/// Abstract base FB for components
{attribute 'reflection' := ''}
FUNCTION_BLOCK ABSTRACT FB_Component IMPLEMENTS ITF_Component

VAR
	/// path of this FB
	{attribute 'no_init' := ''}
	{attribute 'instance-path' := ''}
	sPath						: STRING;	
	/// Unique ID
	nId							: INT;		
	/// component type
	eTyp						: E_ComponentType;
	/// component name
	sName						: STRING;
	/// BMK name
	sBMK						: STRING;
	/// Area
	eMachineArea				: E_MachineArea;			
	
	/// component enable flag
	bEnable						: BOOL := FALSE;
	/// component state
	eState						: E_ComponentState;	
	
	/// Safety
	refEStop					: REFERENCE TO FB_EmergencyStop;
	aitfSafetyComp				: ARRAY[0..COMP.nMaxComponents] OF ITF_SafetyComp;
	bAccessPermit				: BOOL;


	/// Others
	itfEventLog					: ITF_EventLog;
	refSetting					: REFERENCE TO ST_MachineSetting;

	nChangeToggle				: INT;
END_VAR

///
/// 
/// HF/www.asma.at/02.2022
///

PROPERTY AccessPermit : BOOL
GET
AccessPermit := bAccessPermit;
END_GET
END_PROPERTY

/// RunSuper component logic
{attribute 'object_name' := 'Base'}
METHOD Base

VAR
	ni			: INT;
END_VAR
// DEFAULT STATE: set state to running
IF eState = E_ComponentState.ready THEN
	eState := E_ComponentState.running;
END_IF

//Eventlog
IF itfEventLog = 0 THEN
	WriteError(E_Event.eEvent_none, 'HMI Referenz nicht gesetzt!');
	eState := E_ComponentState.error;
	RETURN;
END_IF


Visu();

IF NOT Enable THEN
	RETURN;
END_IF

Run();
END_METHOD

PROPERTY BMK : STRING
GET
BMK := sBMK;
END_GET
SET
sBMK := BMK;
END_SET
END_PROPERTY

METHOD ChangeToggle : BOOL
VAR_INPUT
END_VAR
nChangeToggle := nChangeToggle + 1;
END_METHOD

PROPERTY EmergencyStop : REFERENCE TO FB_EmergencyStop
GET
IF __ISVALIDREF(refEStop) THEN
	EmergencyStop REF= refEStop;
END_IF
END_GET
SET
refEStop REF= EmergencyStop;
END_SET
END_PROPERTY

/// Get's or set's a value indicating whether this component is active or not.
PROPERTY Enable : BOOL
GET
Enable := bEnable;
END_GET
SET
bEnable := Enable;
END_SET
END_PROPERTY

METHOD FB_init : BOOL
VAR_INPUT
	bInitRetains : BOOL := TRUE; // if TRUE, the retain variables are initialized (warm start / cold start)
	bInCopyCode : BOOL := TRUE;  // if TRUE, the instance afterwards gets moved into the copy code (online change)
END_VAR
nId := nId + 1;
itfEventLog := GVL.fbEventLog;
refSetting REF= GVL.stSetting;
refEStop REF= GVL.fbEStop;
Init();
END_METHOD

/// Halt component logic
{attribute 'object_name' := 'Halt'}
METHOD Halt : E_OperationResult

VAR_INPUT
	StoppCategory					: INT;			// 0...ungesteuertes Stillsetzen     1...gesteuertes Stillsetzen     2...gesteuertes Stillsetzen ohne Trennung der Energiezufuhr							
END_VAR
bAccessPermit := TRUE;
END_METHOD

/// Unique component ID (cam be used as index: P_ComponentPool.aComponents[eID]...)
PROPERTY ID : INT
GET
ID := nId;
END_GET
SET
nId := Id;
END_SET
END_PROPERTY

/// Init component logic
{attribute 'object_name' := 'Init'}
METHOD Init : E_OperationResult
END_METHOD

PROPERTY MachineArea : E_MachineArea
GET
MachineArea := eMachineArea;
END_GET
SET
eMachineArea := MachineArea;
END_SET
END_PROPERTY

PROPERTY Name : STRING
GET
Name := sName;
END_GET
SET
sName := Name;
END_SET
END_PROPERTY

PROPERTY Path : String
GET
Path := sPath;
END_GET
END_PROPERTY

METHOD RegisterSafetyComp : BOOL
VAR_INPUT
	SafetyComp				: ITF_SafetyComp;
END_VAR
VAR
	ni						: INT;
END_VAR
FOR ni:= 0 TO COMP.nMaxComponents DO

	IF aitfSafetyComp[ni] = SafetyComp THEN
		RETURN;
	END_IF
	
	IF aitfSafetyComp[ni] <> 0 THEN
		CONTINUE;
	END_IF
	
	aitfSafetyComp[ni] := SafetyComp;
	aitfSafetyComp[ni].RegisterComponent(THIS^);
	RETURN;
	
END_FOR
END_METHOD

/// ResetSuper component logic
{attribute 'object_name' := 'Reset'}
METHOD Reset : E_OperationResult
// DEFAULT STATE: set state to ready
eState := E_ComponentState.ready;
END_METHOD

/// RestartSuper component logic
{attribute 'object_name' := 'Restart'}
METHOD Restart : E_OperationResult
VAR_INPUT
END_VAR
bAccessPermit := FALSE;
END_METHOD

/// RunSuper component logic
{attribute 'object_name' := 'Run'}
METHOD Abstract Run
END_METHOD

PROPERTY SafeEnvironment : BOOL
GET
VAR
	ni				: INT;
END_VAR
SafeEnvironment := TRUE;

FOR ni:= 0 TO COMP.nMaxComponents DO
	
	IF aitfSafetyComp[ni] <> 0 AND_THEN NOT aitfSafetyComp[ni].Safe THEN
		SafeEnvironment := FALSE;
	END_IF

END_FOR
END_GET
END_PROPERTY

/// Get's value representing the component state.
PROPERTY State : E_ComponentState
GET
State := eState;
END_GET
END_PROPERTY

/// Get's value representing the component state.
PROPERTY StateAsString : STRING
GET
CASE eState OF

	E_ComponentState.none :
		StateAsString := 'undefiniert';
	/// Component is resetting
	E_ComponentState.resetting:
		StateAsString := 'wird zurückgesetzt';
	/// Component is ready
	E_ComponentState.ready:
		StateAsString := 'ist bereit';
	/// Component is running
	E_ComponentState.running:
		StateAsString := 'wird ausgeführt';
	/// Component has error
	E_ComponentState.error:
		StateAsString := 'ist fehlerhaft';

END_CASE
END_GET
END_PROPERTY

PROPERTY Typ : E_ComponentType
GET
Typ := eTyp;
END_GET
END_PROPERTY

/// Visu component logic
{attribute 'object_name' := 'Visu'}
METHOD Abstract Visu
END_METHOD

METHOD VisuBase
VAR_IN_OUT
	stCompVisu					: ST_ComponentVisu;
END_VAR
// Visu
stCompVisu.bEnable := bEnable;
stCompVisu.bAccessPermit := AccessPermit;
stCompVisu.bError := eState = E_Componentstate.error;
stCompVisu.bRunning := eState = E_Componentstate.running;
stCompVisu.eState := eState;
stCompVisu.sName := sName;

IF stCompVisu.bReset THEN
	stCompVisu.bReset := FALSE;	
	Reset();
END_IF
END_METHOD

METHOD WriteError
VAR_INPUT
	Event			: E_Event;
	Description 	: T_MaxString;
END_VAR
WriteEvent(ePriority_fault, Event, Description, TRUE);
END_METHOD

METHOD WriteEvent
VAR_INPUT
	Priority		: E_Priority;
	Event			: E_Event;
	Description 	: T_MaxString;
	Signalize		: BOOL;
END_VAR
VAR
	tmpItem: ST_Event;
END_VAR
// chk
IF itfEventLog = 0 THEN
	RETURN;
END_IF

tmpItem.eComponent := eTyp;
tmpItem.eEventID := Event;
tmpItem.eMachineArea := eMachineArea;
tmpItem.sPosition := sBMK;
tmpItem.ePriority := Priority;
tmpItem.nComponentID := nId;
tmpItem.sDescription := Description;
tmpItem.bSignalize := Signalize;
tmpItem.refComponent REF= THIS^;

itfEventLog.SetEvent(tmpItem);
END_METHOD

METHOD WriteInfo
VAR_INPUT
	Event			: E_Event;
	Description 	: T_MaxString;
END_VAR
WriteEvent(ePriority_info, Event, Description, FALSE);
END_METHOD

METHOD WriteWarning
VAR_INPUT
	Event			: E_Event;
	Description 	: T_MaxString;
	Signal			: BOOL;
END_VAR
VAR
	tmpItem			: ST_Event;
END_VAR
WriteEvent(ePriority_warning, Event, Description, Signal);
END_METHOD

END_FUNCTION_BLOCK

(* stored: Version 1.1.0.1
   POU FB_Component: Id {c18f24bd-a664-4b00-87c6-35388a9e2c13}, SpecialFunc None
   Folder Abstract: Id {74ace20b-84be-4a97-82c0-d348ab638f2b}
   Folder Properties: Id {2d8306c8-917b-4b20-9aa7-5415be6cad83}
   Folder Utilities: Id {18cd2ad0-5a5a-4e5f-92e4-b0238b542ab5}
   Property AccessPermit: Id {01de2613-1fdc-4238-9d0f-b61744631c69}
   Get Get: Id {d0f0ca6c-2e80-4b7b-abfc-89db46355afd}
   Method Base: Id {2713eafa-f1d8-4a9a-bf25-6ca9cb07ffb7}
   Property BMK: Id {3e8ee465-5189-4f2f-9d15-0d6a660f5497}
   Get Get: Id {01c92174-19fd-4b80-81d2-175c5750d2bc}
   Set Set: Id {b8ef3cfc-b534-4fcd-97bc-b47816b7b27a}
   Method ChangeToggle: Id {3b0a0586-d96d-42a6-bdb9-f4e6fc39e69e}
   Property EmergencyStop: Id {d611fe1a-6ee7-493e-8715-510afc3d8a9b}
   Get Get: Id {3be43057-3b95-4322-8a51-03383bc7aadd}
   Set Set: Id {c9d09d71-eada-43fe-8284-0a110c5639b3}
   Property Enable: Id {ad08f73b-d076-4ffc-a47f-109b9002f3f0}
   Get Get: Id {8dd8e62e-65cf-4eae-a985-79199664088e}
   Set Set: Id {1d543709-b1d6-4f2d-af6c-97246f4599c2}
   Method FB_init: Id {f2d62d5e-1f23-4c7a-9f92-516abe433c20}
   Method Halt: Id {b88e9e37-d0ce-4cec-931a-fe7e44e673be}
   Property ID: Id {7adf225e-7442-4f77-874e-8de91565912f}
   Get Get: Id {ddac6993-c733-47b1-a445-f075002f8c38}
   Set Set: Id {9987bba1-8297-46ec-8910-10e8ca7a5cd6}
   Method Init: Id {f1064f72-96c7-4897-90d8-0bc004b05e95}
   Property MachineArea: Id {5002829a-7be9-4fd2-bdb1-4f471524ec33}
   Get Get: Id {b1107982-d402-48e8-82e1-34f3ffa3cd58}
   Set Set: Id {3ad4b5e6-3b5e-468e-b88a-52a5ed7a2777}
   Property Name: Id {97507556-cbd6-4656-a4b4-7ef03ea2ff1e}
   Get Get: Id {5bc1be01-8584-43a7-b2c4-089d7b7d1290}
   Set Set: Id {cdf272ad-e29a-4767-ad58-2d41f72fa33a}
   Property Path: Id {f15c3da9-69b6-42be-b750-91438e4fc191}
   Get Get: Id {c3c5d9a1-7c3c-440f-abee-27056ac72a80}
   Method RegisterSafetyComp: Id {51549f56-0d17-4c9e-b529-7b8edc0a6829}
   Method Reset: Id {53e23aa0-51c1-4eb8-a9a2-a57148f04799}
   Method Restart: Id {89d91b38-868a-44ea-bfdd-7a93d6d9b0b1}
   Method Run: Id {bef95d86-7c5e-4a90-8287-2db60c403500}
   Property SafeEnvironment: Id {4797286a-b210-4fd0-a257-36eb9f2ddd9c}
   Get Get: Id {f4d0eabc-a86a-4c8c-a922-4e2d0913b2c3}
   Property State: Id {d68fb6ae-0af8-44c3-bb4d-32b1388481b9}
   Get Get: Id {b4088dcc-e43a-4064-b0df-93c47386d3d2}
   Property StateAsString: Id {bffb55f1-1ef3-4369-ab66-e92ce785efbd}
   Get Get: Id {3dd43a60-ec91-4906-860b-12629fae2ae4}
   Property Typ: Id {987dd2cf-7ace-4cc4-856e-8b41f907e2c3}
   Get Get: Id {9fd10945-acfb-45ad-818f-6e98f300ba25}
   Method Visu: Id {ccb64397-b3bd-44ad-a340-d5df5374177c}
   Method VisuBase: Id {d0c2b612-1946-438d-9cf4-b5c5d137c98e}
   Method WriteError: Id {a92622fe-49fc-4553-8379-a99997764084}
   Method WriteEvent: Id {583be540-6251-46c4-8656-e5b754778d2f}
   Method WriteInfo: Id {c2be943a-77e2-432b-be2b-8003842ed1ca}
   Method WriteWarning: Id {05cae7cb-6c8d-4876-827e-346c099d6a8b} *)
